FUNCTION_BLOCK FB_CraneStatus
VAR_INPUT
	bPower : BOOL;
	bStart : BOOL;
	bStop : BOOL;
	bRunning : BOOL;
	bError : BOOL;
END_VAR
VAR_OUTPUT
	eCraneStatus : E_CraneStatus := E_CraneStatus.PowerOff;
END_VAR
VAR
END_VAR

//Status state machine
CASE eCraneStatus OF
	E_CraneStatus.PowerOff:
		IF bPower THEN
			eCraneStatus := E_CraneStatus.Checking;
		END_IF	
	
	E_CraneStatus.Error:
		IF NOT bError THEN
			eCraneStatus := E_CraneStatus.Checking;
		END_IF
		
	E_CraneStatus.Checking:
		IF (NOT bError) THEN
			eCraneStatus := E_CraneStatus.Ready;
		ELSE
			eCraneStatus := E_CraneStatus.Error;
		END_IF
		
		IF bPower AND NOT bError THEN
			eCraneStatus := E_CraneStatus.Ready;
		ELSE
			eCraneStatus := E_CraneStatus.PowerOff;
		END_IF
		
	E_CraneStatus.Ready:
		IF bStart AND bPower AND NOT(bError) THEN
			HMI.bRunning := TRUE;
			eCraneStatus := E_CraneStatus.Running;
		END_IF	
		
		IF  NOT(bPower) OR bError THEN
			eCraneStatus := E_CraneStatus.Checking;
		END_IF	
		
	E_CraneStatus.Running:
		eCraneStatus := F_CheckPistonPosition();
		IF bStop THEN
			eCraneStatus := E_CraneStatus.Stopping;
		END_IF
		
		IF bError OR NOT bRunning OR NOT bPOWER THEN
			eCraneStatus := E_CraneStatus.Checking;
		END_IF
		
	E_CraneStatus.Stopping:
		HMI.bRunning := FALSE;
		HMI.bStart := FALSE;
	
		IF NOT bRunning OR bPower OR bError THEN
			eCraneStatus := E_CraneStatus.Checking;
		END_IF
		
	ELSE
		eCraneStatus := E_CraneStatus.Checking;
		
END_CASE

END_FUNCTION_BLOCK

(* stored: Version 1.1.0.1, ProductVersion 3.1.4024.10
   POU FB_CraneStatus: Id {329bc91d-7383-4ae4-a297-132803e3e6a7}, SpecialFunc None *)
